# EPICS substitutions: iocBoot/ioc13ida/ipUnidig.substitutions
# Set the SCAN field of the longin record and bi record #0 to "1 second", rather than I/O
# interrupt, because the quadEM toggles input #0 at 800Hz, and that is too much load on the IOC

file "$(IPUNIDIG)/db/IpUnidigLi.db"
{
pattern
{P,       R,          PORT,       SCAN}
{13IDA:,  Unidig1Li,  Unidig1, "1 second"}
}

file "$(IPUNIDIG)/db/IpUnidigBi.db"
{
pattern
{P,       R,          PORT,    MASK,        SCAN}
{13IDA:, Unidig1Bi0,  Unidig1, 0x000001, "1 second"}
{13IDA:, Unidig1Bi1,  Unidig1, 0x000002, "I/O Intr"}
{13IDA:, Unidig1Bi2,  Unidig1, 0x000004, "I/O Intr"}
{13IDA:, Unidig1Bi3,  Unidig1, 0x000008, "I/O Intr"}
{13IDA:, Unidig1Bi4,  Unidig1, 0x000010, "I/O Intr"}
{13IDA:, Unidig1Bi5,  Unidig1, 0x000020, "I/O Intr"}
{13IDA:, Unidig1Bi6,  Unidig1, 0x000040, "I/O Intr"}
{13IDA:, Unidig1Bi7,  Unidig1, 0x000080, "I/O Intr"}
{13IDA:, Unidig1Bi8,  Unidig1, 0x000100, "I/O Intr"}
{13IDA:, Unidig1Bi9,  Unidig1, 0x000200, "I/O Intr"}
{13IDA:, Unidig1Bi10, Unidig1, 0x000400, "I/O Intr"}
{13IDA:, Unidig1Bi11, Unidig1, 0x000800, "I/O Intr"}
{13IDA:, Unidig1Bi12, Unidig1, 0x001000, "I/O Intr"}
{13IDA:, Unidig1Bi13, Unidig1, 0x002000, "I/O Intr"}
{13IDA:, Unidig1Bi14, Unidig1, 0x004000, "I/O Intr"}
{13IDA:, Unidig1Bi15, Unidig1, 0x008000, "I/O Intr"}
{13IDA:, Unidig1Bi16, Unidig1, 0x010000, "I/O Intr"}
{13IDA:, Unidig1Bi17, Unidig1, 0x020000, "I/O Intr"}
{13IDA:, Unidig1Bi18, Unidig1, 0x040000, "I/O Intr"}
{13IDA:, Unidig1Bi19, Unidig1, 0x080000, "I/O Intr"}
{13IDA:, Unidig1Bi20, Unidig1, 0x100000, "I/O Intr"}
{13IDA:, Unidig1Bi21, Unidig1, 0x200000, "I/O Intr"}
{13IDA:, Unidig1Bi22, Unidig1, 0x400000, "I/O Intr"}
{13IDA:, Unidig1Bi23, Unidig1, 0x800000, "I/O Intr"}
}

file "$(IPUNIDIG)/db/IpUnidigBo.db"
{
pattern
{P,       R,          PORT,    MASK}
{13IDA:, Unidig1Bo0,  Unidig1, 0x000001}
{13IDA:, Unidig1Bo1,  Unidig1, 0x000002}
{13IDA:, Unidig1Bo2,  Unidig1, 0x000004}
{13IDA:, Unidig1Bo3,  Unidig1, 0x000008}
{13IDA:, Unidig1Bo4,  Unidig1, 0x000010}
{13IDA:, Unidig1Bo5,  Unidig1, 0x000020}
{13IDA:, Unidig1Bo6,  Unidig1, 0x000040}
{13IDA:, Unidig1Bo7,  Unidig1, 0x000080}
{13IDA:, Unidig1Bo8,  Unidig1, 0x000100}
{13IDA:, Unidig1Bo9,  Unidig1, 0x000200}
{13IDA:, Unidig1Bo10, Unidig1, 0x000400}
{13IDA:, Unidig1Bo11, Unidig1, 0x000800}
{13IDA:, Unidig1Bo12, Unidig1, 0x001000}
{13IDA:, Unidig1Bo13, Unidig1, 0x002000}
{13IDA:, Unidig1Bo14, Unidig1, 0x004000}
{13IDA:, Unidig1Bo15, Unidig1, 0x008000}
{13IDA:, Unidig1Bo16, Unidig1, 0x010000}
{13IDA:, Unidig1Bo17, Unidig1, 0x020000}
{13IDA:, Unidig1Bo18, Unidig1, 0x040000}
{13IDA:, Unidig1Bo19, Unidig1, 0x080000}
{13IDA:, Unidig1Bo20, Unidig1, 0x100000}
{13IDA:, Unidig1Bo21, Unidig1, 0x200000}
{13IDA:, Unidig1Bo22, Unidig1, 0x400000}
{13IDA:, Unidig1Bo23, Unidig1, 0x800000}
}

file "$(IPUNIDIG)/db/IpUnidigLo.db"
{
pattern
{P,       R,          PORT}
{13IDA:,  Unidig1Lo,  Unidig1}
}
